FUNCTION_BLOCK ProduceTemperaturePayload (* Produce IndoorTemperature payload *)
  (* Standard: 61499-2; Description: Copyright (c) 2018 fortiss GmbH This program and the accompanying materials are made available under the terms of the Eclipse Public License 2.0 which is available at https://www.eclipse.org/legal/epl-2.0/ SPDX-License-Identifier: EPL-2.0 *)
  (* Version 1.0, 2018-09-21, Jose Cabral, fortiss GmbH *)
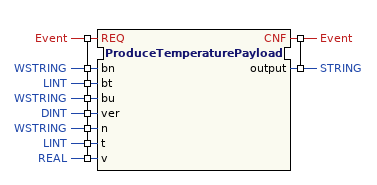
  EVENT_INPUT
    REQ WITH bu, v, t, n, bt, bn, ver; (* Produce Payload *)
  END_EVENT
  EVENT_OUTPUT
    CNF WITH output; (* Payload produced *)
  END_EVENT
  VAR_INPUT
    bn : WSTRING; (* Base Name, this field stores the name of the ArrowheadSystem *)
    bt : LINT; (* Base Time, this field contains the unix timestamp of the sensor readout *)
    bu : WSTRING; (* Base Unit of the sensor readout *)
    ver : DINT; (* Version identifier *)
    n : WSTRING; (* Name of the temperature *)
    t : LINT; (* time of the value *)
    v : REAL; (* value *)
  END_VAR
  VAR_OUTPUT
    output : STRING; (* Result payload *)
  END_VAR
END_FUNCTION_BLOCK
